Staubli VAL3: addAction.pgx

public program addAction(ActionItem& x_aAction[])
  local num l_nSizeAction
  local num l_nSize
  local num l_nIndex
begin
  // mutex it
  setMutex(bActionMutex)
  //
  // insert a new action
  //
  if aAction.iInstr.sType!="null"
    append(aAction)
  endIf
  // set the size
  l_nSizeAction=size(aAction)-1
  // copy it
  aAction[l_nSizeAction]=x_aAction
  // update the nMoveId...
  l_nSize=size(tTrajCycle)-1
  l_nIndex=min(x_aAction.nPointId,size(tTrajCycle[l_nSize].tSuper)-1)
  tTrajCycle[l_nSize].tSuper[l_nIndex].nMoveId=x_aAction.nMoveId
  // release
  bActionMutex=false
end
